// TIA Portal V19 export
FUNCTION "FC_FW_Auftrag_Step3_KB" : Void   // FC1083, LAD
TITLE = Schritt CM03 -> CM03 CM04-> CM04
{ S7_Optimized_Access := 'TRUE' }
// Ältesten Warenträger in CM03 / CM04 suchen und wieder einsetzen
// stored: AutoNumber false, SetENOAutomatically false
   VAR_INPUT
      Frg_Schritt : Bool;
   END_VAR
   VAR_OUTPUT
      nextStep : Bool;
      startStep : Bool;
      parkStep : Bool;
   END_VAR
   VAR_IN_OUT
      Quelle : Int;
      Ziel : Int;
      Positionen : Array[1..30] of "UDT_Auftrag_Pos";
   END_VAR
   VAR_TEMP
      Sperre_Kurz_li : Bool;
      Sperre_Kurz_re : Bool;
      Sperre_Lang : Bool;
      Vorzug : Bool;
      Befehl_ok : Bool;
      tmpQuelle : Int;
      Oldest : Real;
   END_VAR
   VAR CONSTANT
      Wt_Cmd_Spuele_CM03 : Int := 7;
      Wt_Cmd_Spuele_CM04 : Int := 19;
   END_VAR
BEGIN

REGION Network 1 (SCL)
   IF (#Quelle <> 0) AND (#Ziel <> 0) THEN
       #nextStep := #Positionen[#Quelle].Sperre;
       #startStep := NOT #nextStep;
       #Quelle := 0;
       #Ziel := 0;
       RETURN;
   END_IF;

   #Quelle := 0;
   #Ziel := 0;
   #nextStep := FALSE;
   #startStep := FALSE;

   IF NOT #Frg_Schritt THEN
       #nextStep := TRUE;
       RETURN;
   END_IF;
END_REGION

REGION Network 2 (SCL): Positionen sperren
   //Groß links nicht möglich
   #Positionen[9].CheckSperre := #Positionen[9].Wt_Cmd <> #Wt_Cmd_Spuele_CM03;

   //Groß rechts nicht möglich
   #Positionen[10].CheckSperre := #Positionen[10].Wt_Cmd <> #Wt_Cmd_Spuele_CM03;

   //Platz spielt keine Rolle, nur CMD

   //Lang in P7
   //-> P8 sperren
   #Positionen[8].CheckSperre := (#Positionen[7].Wt_Typ = "WT_Typ_LS") OR (#Positionen[8].Wt_Cmd <> #Wt_Cmd_Spuele_CM03);

   //-> P7 sperren
   #Positionen[7].CheckSperre := (#Positionen[7].Wt_Cmd <> #Wt_Cmd_Spuele_CM03);

   //Lang in P11 
   //-> P12 sperren
   #Positionen[12].CheckSperre := (#Positionen[11].Wt_Typ = "WT_Typ_LS") OR (#Positionen[12].Wt_Cmd <> #Wt_Cmd_Spuele_CM03);

   //Lang in P11
   //-> P11 sperren
   #Positionen[11].CheckSperre := (#Positionen[11].Wt_Cmd <> #Wt_Cmd_Spuele_CM03);

   //Lang in P19
   //-> P20 sperren
   #Positionen[20].CheckSperre := (#Positionen[19].Wt_Typ = "WT_Typ_LS") OR (#Positionen[20].Wt_Cmd <> #Wt_Cmd_Spuele_CM04);

   //-> P19 sperren
   #Positionen[19].CheckSperre := (#Positionen[19].Wt_Cmd <> #Wt_Cmd_Spuele_CM04);

   //Lang in P23 
   //-> P24 sperren
   #Positionen[24].CheckSperre := (#Positionen[23].Wt_Typ = "WT_Typ_LS") OR (#Positionen[24].Wt_Cmd = #Wt_Cmd_Spuele_CM04);

   //Lang in P23
   //-> P23 sperren
   #Positionen[23].CheckSperre := (#Positionen[23].Wt_Cmd <> #Wt_Cmd_Spuele_CM04);
END_REGION

REGION Network 3 (SCL): Ältesten WT suchen
   //
   #Oldest := 0;
   #tmpQuelle := 0;

   //CM03
   "FC_FW_Auftrag_Suche"(Pos1 := 7,
                         Pos2 := 12,
                         Positionen := #Positionen,
                         Quelle := #tmpQuelle,
                         Oldest := #Oldest);

   //CM04
   "FC_FW_Auftrag_Suche"(Pos1 := 19,
                         Pos2 := 24,
                         Positionen := #Positionen,
                         Quelle := #tmpQuelle,
                         Oldest := #Oldest);
END_REGION

REGION Network 4 (SCL): Auswertung
   IF #tmpQuelle = 0 THEN
       //kein WT
       #nextStep := TRUE;
       RETURN;
   END_IF;

   IF NOT #Positionen[#tmpQuelle].Fertig THEN
       #parkStep := TRUE;
       RETURN;
   END_IF;

   IF (#tmpQuelle = 9) THEN
       //Gross links - nur 161

           "FC_FW_Auftrag_Befehl"(inQuelle := #tmpQuelle,
                                  inZiel := 9,
                                  Befehl_ok => #Befehl_ok,
                                  outQuelle => #Quelle,
                                  outZiel => #Ziel);

           #nextStep := NOT #Befehl_ok;

       RETURN;
   END_IF;

   IF (#tmpQuelle = 10) THEN
       //Gross rechts - nur "161"

           "FC_FW_Auftrag_Befehl"(inQuelle := #tmpQuelle,
                                  inZiel := 10,
                                  Befehl_ok => #Befehl_ok,
                                  outQuelle => #Quelle,
                                  outZiel => #Ziel);

           #nextStep := NOT #Befehl_ok;

       RETURN;
   END_IF;

   IF (#Positionen[#tmpQuelle].Wt_Typ = "WT_Typ_LS") AND (#tmpQuelle = 7) THEN
       //Lang "161"
       "FC_FW_Auftrag_Befehl"(inQuelle := #tmpQuelle,
                                  inZiel := 7,
                                  Befehl_ok => #Befehl_ok,
                                  outQuelle => #Quelle,
                                  outZiel => #Ziel);

           #nextStep := NOT #Befehl_ok;

        RETURN;
   END_IF;


   IF (#Positionen[#tmpQuelle].Wt_Typ = "WT_Typ_LS") AND (#tmpQuelle = 11) THEN
       //Lang "161"
       "FC_FW_Auftrag_Befehl"(inQuelle := #tmpQuelle,
                              inZiel := 11,
                              Befehl_ok => #Befehl_ok,
                              outQuelle => #Quelle,
                              outZiel => #Ziel);

       #nextStep := NOT #Befehl_ok;

       RETURN;
   END_IF;

   IF (#Positionen[#tmpQuelle].Wt_Typ = "WT_Typ_LS") AND (#tmpQuelle = 19) THEN
       //Lang "151"
       "FC_FW_Auftrag_Befehl"(inQuelle := #tmpQuelle,
                              inZiel := 19,
                              Befehl_ok => #Befehl_ok,
                              outQuelle => #Quelle,
                              outZiel => #Ziel);

       #nextStep := NOT #Befehl_ok;

       RETURN;
   END_IF;


   IF (#Positionen[#tmpQuelle].Wt_Typ = "WT_Typ_LS") AND (#tmpQuelle = 23) THEN
       //Lang "151"
       "FC_FW_Auftrag_Befehl"(inQuelle := #tmpQuelle,
                              inZiel := 23,
                              Befehl_ok => #Befehl_ok,
                              outQuelle => #Quelle,
                              outZiel => #Ziel);

       #nextStep := NOT #Befehl_ok;

       RETURN;
   END_IF;


   IF (#tmpQuelle = 7) THEN
       //Kurz links "161
       "FC_FW_Auftrag_Befehl"(inQuelle := #tmpQuelle,
                                  inZiel := 7,
                                  Befehl_ok => #Befehl_ok,
                                  outQuelle => #Quelle,
                                  outZiel => #Ziel);

           #nextStep := NOT #Befehl_ok;
           RETURN;
   END_IF;

   IF (#tmpQuelle = 11) THEN
       //Kurz links "161
       "FC_FW_Auftrag_Befehl"(inQuelle := #tmpQuelle,
                              inZiel := 11,
                              Befehl_ok => #Befehl_ok,
                              outQuelle => #Quelle,
                              outZiel => #Ziel);

       #nextStep := NOT #Befehl_ok;
       RETURN;
   END_IF;

   IF (#tmpQuelle = 8) THEN
       //Kurz rechtss "161
       "FC_FW_Auftrag_Befehl"(inQuelle := #tmpQuelle,
                              inZiel := 8,
                              Befehl_ok => #Befehl_ok,
                              outQuelle => #Quelle,
                              outZiel => #Ziel);

       #nextStep := NOT #Befehl_ok;
       RETURN;
   END_IF;

   IF (#tmpQuelle = 12) THEN
       //Kurz rechts "161
       "FC_FW_Auftrag_Befehl"(inQuelle := #tmpQuelle,
                              inZiel := 12,
                              Befehl_ok => #Befehl_ok,
                              outQuelle => #Quelle,
                              outZiel => #Ziel);

       #nextStep := NOT #Befehl_ok;
       RETURN;
   END_IF;


   IF (#tmpQuelle = 19) THEN
       //Kurz links "151
       "FC_FW_Auftrag_Befehl"(inQuelle := #tmpQuelle,
                              inZiel := 19,
                              Befehl_ok => #Befehl_ok,
                              outQuelle => #Quelle,
                              outZiel => #Ziel);

       #nextStep := NOT #Befehl_ok;
       RETURN;
   END_IF;

   IF (#tmpQuelle = 23) THEN
       //Kurz links "151
       "FC_FW_Auftrag_Befehl"(inQuelle := #tmpQuelle,
                              inZiel := 23,
                              Befehl_ok => #Befehl_ok,
                              outQuelle => #Quelle,
                              outZiel => #Ziel);

       #nextStep := NOT #Befehl_ok;
       RETURN;
   END_IF;

   IF (#tmpQuelle = 20) THEN
       //Kurz rechtss "151
       "FC_FW_Auftrag_Befehl"(inQuelle := #tmpQuelle,
                              inZiel := 20,
                              Befehl_ok => #Befehl_ok,
                              outQuelle => #Quelle,
                              outZiel => #Ziel);

       #nextStep := NOT #Befehl_ok;
       RETURN;
   END_IF;

   IF (#tmpQuelle = 24) THEN
       //Kurz rechts "151
       "FC_FW_Auftrag_Befehl"(inQuelle := #tmpQuelle,
                              inZiel := 24,
                              Befehl_ok => #Befehl_ok,
                              outQuelle => #Quelle,
                              outZiel => #Ziel);

       #nextStep := NOT #Befehl_ok;
       RETURN;
   END_IF;
   //
   #nextStep := TRUE;
END_REGION
END_FUNCTION
